Staubli VAL3: setSAM.pgx

program setSAM(string messageBuffer (dimensions=1), string message (dimensions=1), num sio_ID (dimensions=1))
  local num indexX
  local num indexY
  local num indexZ
  local bool isnum
  local num samX
  local num samY
  local num samZ
begin
  putln(messageBuffer)
  currentPickPosJ=herej()
  currentPickPos=jointToPoint(flange,world,currentPickPosJ)
  //numXold=numXarray
  //numYold=numYarray
  indexX=find(messageBuffer,("#Y"))
  indexZ=find(messageBuffer,("#Z"))
  toNum(left(messageBuffer,indexX),samX,isnum)
  if isnum==false
    taskCreate "sendStatus",10,sendStatus("... X is not a number ...",sio_ID)
    putln("... X is not a number ...")
  endIf
  indexY=len(messageBuffer)-find(messageBuffer,("#Z"))-2
  toNum(right(messageBuffer,indexY),samY,isnum)
  if isnum==false
    taskCreate "sendStatus",10,sendStatus("... Y is not a number ...",sio_ID)
    putln("... Y is not a number ...")
  endIf
  toNum(mid(messageBuffer,indexZ-indexY,indexY+2),samZ,isnum)
  if isnum==false
    taskCreate "sendStatus",10,sendStatus("... Z is not a number ...",sio_ID)
    putln("... Z is not a number ...")
  endIf
  putln("show sam values:")
  putln(toString(".3",samX))
  putln(toString(".3",samY))
  putln(toString(".3",samZ))
  movel(appro(currentPickPos,{samY,-samX,-samZ,0,0,0}),flange,mNomSpeed)
  waitEndMove()
  taskCreate "sendStatus",10,sendStatus(message,sio_ID)
  putln(message)
  //required shape: e.g. 'setSAM#X1.12345#Y2.3456#Z0.2345'
end
